Universal Robots PolyScope program: Main.urp

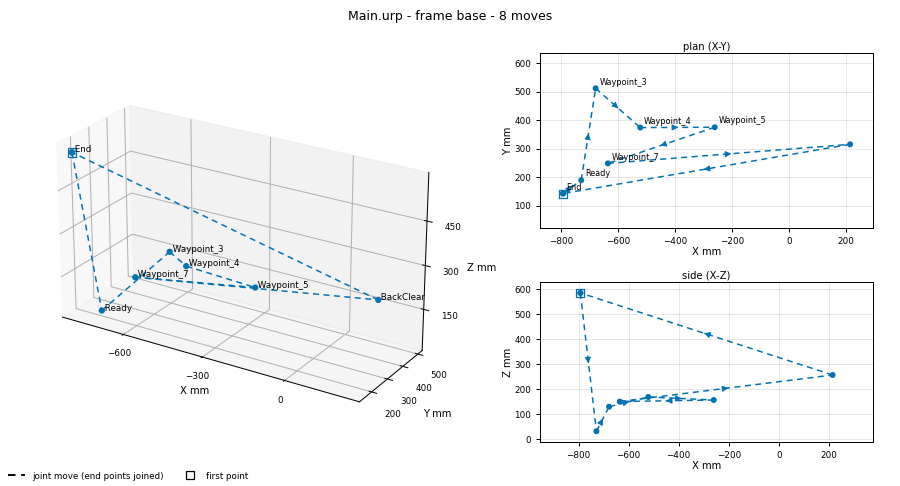
[picture p0: tool path of Main.urp in frame base, 8 of 8 moves have a stored position in this frame; points joined in program order, loops and branches not executed]
Program Main (installation=default directory=/programs/new folder createdIn=5.11.5.1010327 lastSavedIn=5.11.5.1010327 robotSerialNumber=20215500677)
Calibrated DH parameters: a=[0.000204, -0.239222, -0.391845, -0.000001, 0.000022, 0]; d=[0.162722, -355.808559, 353.37206, 2.570385, 0.099741, 0.099629]; alpha=[1.571124, 0.000988, 0.008295, 1.568963, -1.570303, 0]; deltaTheta=[0, -0.973091, 7.204745, 0.05153, 0, 0]
InitVariablesNode variables(variable(name=count, expression=0))
Robot Program (runOnlyOnce=false)
  count := count+1
  Loop Forever
    Wait DigitalInput pin=digital_in[0]; digitalValue=1
    Set DigitalOutput tcp=Dynabrade1; pin=digital_out[1]; digitalValue=1
    MoveJ speed 60 deg/s, acceleration 80 deg/s^2 (useActiveTCP=true) feature=Point_1
      Waypoint End: TCP in base x=-792.986 y=142.126 z=584.824 mm, rx=0.6139 ry=-1.4821 rz=-0.614 rad; joints [333.592, -61.672, 69.104, -187.689, -63.582, 225.626] deg; TCP offset x=0 y=0 z=105 mm, rx=0 ry=0 rz=0 rad; feature pose in base x=-675 y=184.662 z=50 mm, rx=0.0001 ry=0 rz=3.1416 rad
    MoveJ speed 60 deg/s, acceleration 80 deg/s^2 (useActiveTCP=false) tcp=Dynabrade1; feature=Point_1
      Waypoint Ready: TCP in base x=-728.914 y=189 z=32.379 mm, rx=0 ry=-3.1416 rz=0 rad; joints [335.226, -42.704, 75.581, -122.851, -89.577, 245.512] deg; TCP offset x=0 y=0 z=105 mm, rx=0 ry=0 rz=0 rad; feature pose in base x=-728.914 y=189 z=30.379 mm, rx=0 ry=0 rz=3.1416 rad
    Call sandTop
    Call positionFace1
    Call sandFace
    MoveJ speed 60 deg/s, acceleration 80 deg/s^2 (useActiveTCP=true) feature=Point_1
      Waypoint Waypoint_3: TCP in base x=-678.243 y=511.665 z=130.309 mm, rx=-1.5708 ry=0 rz=0 rad; joints [325.381, -29.88, 51.308, -20.942, 145.47, 180.61] deg; TCP offset x=0 y=0 z=105 mm, rx=0 ry=0 rz=0 rad
    Call sandFace
    MoveJ speed 60 deg/s, acceleration 80 deg/s^2 (useActiveTCP=true) feature=Point_1
      Waypoint Waypoint_4: TCP in base x=-521.6 y=373.868 z=169.065 mm, rx=-0.0271 ry=3.1414 rz=-0.0001 rad; joints [312.325, -65.395, 91.797, -116.371, -89.573, 221.581] deg; TCP offset x=0 y=0 z=105 mm, rx=0 ry=0 rz=0 rad
      Waypoint Waypoint_5: TCP in base x=-259.991 y=375 z=156.997 mm, rx=-0.4232 ry=1.5359 rz=-0.398 rad; joints [308.406, -51.401, 88.304, -38.01, -142.187, 238.952] deg; TCP offset x=0 y=0 z=105 mm, rx=0 ry=0 rz=0 rad; feature pose in base x=-585 y=315 z=57 mm, rx=0.0001 ry=0 rz=3.1416 rad
    Call sandFace_1
    URCap Finishing Tool Control (Robotiq_Copilot, Robotiq Inc.) dataModel(FinishingToolStateKey=false, ToolOutputNameKey=digital_out[0], HackTriggeringContributionIsDefinedMethodKey=true)
    MoveJ speed 60 deg/s, acceleration 80 deg/s^2 (useActiveTCP=true) feature=Base
      Waypoint Waypoint_7: TCP in base x=-635.269 y=248.035 z=150.92 mm, rx=-0.4354 ry=3.0052 rz=-0.0196 rad; joints [328.369, -57.223, 80.615, -108.259, -92.837, 222.208] deg; TCP offset x=0 y=0 z=105 mm, rx=0 ry=0 rz=0 rad
    MoveJ speed 60 deg/s, acceleration 80 deg/s^2 (useActiveTCP=true) feature=Point_1
      Waypoint BackClear: TCP in base x=215.017 y=314.968 z=256.959 mm, rx=2.2214 ry=2.2214 rz=0.0002 rad; joints [215.107, -106.327, 122.312, -105.964, -89.576, 215.301] deg; TCP offset x=0 y=0 z=105 mm, rx=0 ry=0 rz=0 rad; feature pose in base x=-585 y=315 z=57 mm, rx=0.0001 ry=0 rz=3.1416 rad
    Call sandBack
    MoveJ speed 60 deg/s, acceleration 80 deg/s^2 (useActiveTCP=true) feature=Point_1
      Waypoint End: TCP in base x=-792.986 y=142.126 z=584.824 mm, rx=0.6139 ry=-1.4821 rz=-0.614 rad; joints [333.592, -61.672, 69.104, -187.689, -63.582, 225.626] deg; TCP offset x=0 y=0 z=105 mm, rx=0 ry=0 rz=0 rad; feature pose in base x=-675 y=184.662 z=50 mm, rx=0.0001 ry=0 rz=3.1416 rad
    Set DigitalOutput tcp=Dynabrade1; pin=digital_out[1]; digitalValue=0
  If count≟20
    Popup Message (haltProgram=false message=change sand paper inputType=Text)
    count := count+1
Event  expression=digital_in[1]≠ True
  Set DigitalOutput tcp=Dynabrade1; pin=digital_out[0]; digitalValue=0
  Set DigitalOutput tcp=Dynabrade1; pin=digital_out[1]; digitalValue=0
  Halt
SubProgram  [hidden by the author, left out]
SubProgram -> sandFace
SubProgram -> sandFace_1
SubProgram -> sandTop
SubProgram -> sandBack
SubProgram sandTop (keepSynchronizedWithDisk=true) programFile=/programs/new folder/sandTop.urp
  MoveL speed 100 mm/s, acceleration 1200 mm/s^2 (useActiveTCP=true) feature=Base
    MoveDirectionNode (selectedDirection=ZPlus) feature=Joint_6_name
      Until TOOL_CONTACT_DETECTION (allowActions=false retraction=0 decelerationAcceleration=3 decelerationAngularAcceleration=34.906585)
  URCap Finishing Tool Control (Robotiq_Copilot, Robotiq Inc.) dataModel(ToolOutputNameKey=digital_out[0], HackTriggeringContributionIsDefinedMethodKey=true)
  Wait Sleep waitTime=2
  URCap Find Surface (Robotiq_Copilot, Robotiq Inc.) dataModel(NodeInitializedKey=true, ZeroSensorBeforeKey=true, WaitForSteadyWrenchOptionKey=false, ls_force=10.0, ls_distance=100.0, ls_speed=5.0, ls_if_distance=false, ls_if_force=false); state(isChildrenLocked=true)
    'Add Stop conditions from the Find Surface node'
  Force Simple feature=Joint_6_name; selection=[0, 0, 1, 0, 0, 0]; wrench=[0, 0, 2, 0, 0, 0]; limitsForce=[0.15, 0.15, 0.15, 1.047198, 1.047198, 1.047198]; limitsMotion=[0.1, 0.1, 0.1, 0.349066, 0.349066, 0.349066]
    MoveL speed 60 mm/s, acceleration 1200 mm/s^2 (useActiveTCP=true) feature=Base
      MoveDirectionNode (selectedDirection=YPlus)
        Until DISTANCE (allowActions=false deceleration=3 distanceNodeType=BLEND) Distance=0.35; motionParameters(blendRadius=0.005)
      MoveDirectionNode (selectedDirection=XPlus)
        Until DISTANCE (allowActions=false deceleration=3 distanceNodeType=BLEND) Distance=0.36; motionParameters(blendRadius=0.005)
      MoveDirectionNode (selectedDirection=YMinus)
        Until DISTANCE (allowActions=false deceleration=3 distanceNodeType=BLEND) Distance=0.35; motionParameters(blendRadius=0.005)
      MoveDirectionNode (selectedDirection=XMinus)
        Until DISTANCE (allowActions=false deceleration=3 distanceNodeType=STOP) Distance=0.36; motionParameters(blendRadius=0.005)
  MoveL speed 60 mm/s, acceleration 1200 mm/s^2 (useActiveTCP=true) feature=Base
    MoveDirectionNode (selectedDirection=ZPlus)
      Until DISTANCE (allowActions=false deceleration=3 distanceNodeType=STOP) Distance=0.025; motionParameters(blendRadius=0)
  URCap Finishing Tool Control (Robotiq_Copilot, Robotiq Inc.) dataModel(ToolOutputNameKey=digital_out[0], FinishingToolStateKey=false, HackTriggeringContributionIsDefinedMethodKey=true)
SubProgram positionFace1 [hidden by the author, left out]
SubProgram sandFace (keepSynchronizedWithDisk=false)
  MoveL speed 250 mm/s, acceleration 1200 mm/s^2 (useActiveTCP=true) feature=Base
    MoveDirectionNode (selectedDirection=ZMinus)
      Until DISTANCE (allowActions=false deceleration=3 distanceNodeType=STOP) Distance=0.072; motionParameters(blendRadius=0)
  MoveL speed 15 mm/s, acceleration 1200 mm/s^2 (useActiveTCP=true) feature=Base
    MoveDirectionNode (selectedDirection=ZPlus) feature=Joint_6_name
      Until TOOL_CONTACT_DETECTION (allowActions=false retraction=0 decelerationAcceleration=3 decelerationAngularAcceleration=34.906585)
    URCap Finishing Tool Control (Robotiq_Copilot, Robotiq Inc.) dataModel(ToolOutputNameKey=digital_out[0], HackTriggeringContributionIsDefinedMethodKey=true)
    Wait Sleep waitTime=2
    URCap Force Control (Robotiq_Copilot, Robotiq Inc.) dataModel(NodeInitializedKey=true, force_x=0, force_y=0, force_mx=0, force_my=0, force_mz=0, limit_x_neg=-100, limit_y_neg=-100, limit_z_neg=-100, limit_x_pos=100, limit_y_pos=100, limit_z_pos=100, limit_mx_neg=-20, limit_my_neg=-20, limit_mz_neg=-20, limit_mx_pos=20, limit_my_pos=20, limit_mz_pos=20, ft_control_x=false, ft_control_y=false, ft_control_mx=false, ft_control_my=false, ft_control_mz=false, stiffness_x=100, stiffness_y=100, stiffness_z_position=100, stiffness_mx=100, stiffness_my=100, stiffness_mz=100, adaptive_stiffness=true, is_force_control_about_actual_position=true, ft_control_z=true, force_z=1, HackTriggeringContributionIsDefinedMethodKey=true, TranslatableFeatureKey=1)
      URCap Force Event (Robotiq_Copilot, Robotiq Inc.) dataModel(NodeInitializedKey=true, NodeTitleKey=Force Event, InteractIfTimeoutOptionKey=false, InteractIfTimeoutNodeInsertedKey=false, InteractTimeoutKey=30, ForceReachedIfTimeoutOptionKey=false, ForceReachedIfTimeoutNodeInsertedKey=false, ForceReachedTimeoutKey=30, IfNotClickedOptionKey=false, IfNotClickedNodeInsertedKey=false, ForceDropRadioButtonKey=true, TorqueDropRadioButtonKey=false, ForceDropKey=10.0, TorqueDropKey=1.0, IsAddSingleTapButtonEnabledKey=true, IsAddDoubleTapButtonEnabledKey=true, AreDuplicatedTapNodesInTreeKey=false, SelectedForceEventKey=2, HackTriggeringContributionIsDefinedMethodKey=true); state(isChildrenLocked=true)
        'Wait until force and torque are reached.'
    MoveDirectionNode (selectedDirection=XPlus) feature=Joint_6_name
      Until DISTANCE (allowActions=false deceleration=3 distanceNodeType=STOP) Distance=0.26; motionParameters(blendRadius=0)
    SuppressedNode
      URCap Find Surface (Robotiq_Copilot, Robotiq Inc.) dataModel(NodeInitializedKey=true, ZeroSensorBeforeKey=true, WaitForSteadyWrenchOptionKey=false, ls_force=10.0, ls_distance=100.0, ls_speed=5.0, ls_if_distance=false, ls_if_force=false); state(isChildrenLocked=true)
        'Add Stop conditions from the Find Surface node'
    SuppressedNode
      Force Simple feature=Joint_6_name; selection=[0, 0, 1, 0, 0, 0]; wrench=[0, 0, 1, 0, 0, 0]; limitsForce=[0.15, 0.15, 0.15, 1.047198, 1.047198, 1.047198]; limitsMotion=[0.1, 0.1, 0.1, 0.349066, 0.349066, 0.349066]
        Placeholder
    URCap Finishing Tool Control (Robotiq_Copilot, Robotiq Inc.) dataModel(FinishingToolStateKey=false, ToolOutputNameKey=digital_out[0], HackTriggeringContributionIsDefinedMethodKey=true)
    MoveDirectionNode (selectedDirection=ZPlus)
      Until DISTANCE (allowActions=false deceleration=3 distanceNodeType=STOP) Distance=0.05; motionParameters(blendRadius=0)
SubProgram sandFace_1 (keepSynchronizedWithDisk=false)
  MoveL speed 250 mm/s, acceleration 1200 mm/s^2 (useActiveTCP=true) feature=Base
    MoveDirectionNode (selectedDirection=ZMinus)
      Until DISTANCE (allowActions=false deceleration=3 distanceNodeType=STOP) Distance=0.072; motionParameters(blendRadius=0)
  MoveL speed 30 mm/s, acceleration 1200 mm/s^2 (useActiveTCP=true) feature=Base
    MoveDirectionNode (selectedDirection=ZPlus) feature=Joint_6_name
      Until TOOL_CONTACT_DETECTION (allowActions=false retraction=0.001 decelerationAcceleration=3 decelerationAngularAcceleration=34.906585)
    URCap Finishing Tool Control (Robotiq_Copilot, Robotiq Inc.) dataModel(ToolOutputNameKey=digital_out[0], HackTriggeringContributionIsDefinedMethodKey=true)
    Wait Sleep waitTime=2
    URCap Force Control (Robotiq_Copilot, Robotiq Inc.) dataModel(NodeInitializedKey=true, force_x=0, force_y=0, force_mx=0, force_my=0, force_mz=0, limit_x_neg=-100, limit_y_neg=-100, limit_z_neg=-100, limit_x_pos=100, limit_y_pos=100, limit_z_pos=100, limit_mx_neg=-20, limit_my_neg=-20, limit_mz_neg=-20, limit_mx_pos=20, limit_my_pos=20, limit_mz_pos=20, ft_control_x=false, ft_control_y=false, ft_control_mx=false, ft_control_my=false, ft_control_mz=false, stiffness_x=100, stiffness_y=100, stiffness_z_position=100, stiffness_mx=100, stiffness_my=100, stiffness_mz=100, adaptive_stiffness=true, is_force_control_about_actual_position=true, ft_control_z=true, force_z=1, HackTriggeringContributionIsDefinedMethodKey=true, TranslatableFeatureKey=1)
      URCap Force Event (Robotiq_Copilot, Robotiq Inc.) dataModel(NodeInitializedKey=true, NodeTitleKey=Force Event, InteractIfTimeoutOptionKey=false, InteractIfTimeoutNodeInsertedKey=false, InteractTimeoutKey=30, ForceReachedIfTimeoutOptionKey=false, ForceReachedIfTimeoutNodeInsertedKey=false, ForceReachedTimeoutKey=30, IfNotClickedOptionKey=false, IfNotClickedNodeInsertedKey=false, ForceDropRadioButtonKey=true, TorqueDropRadioButtonKey=false, ForceDropKey=10.0, TorqueDropKey=1.0, IsAddSingleTapButtonEnabledKey=true, IsAddDoubleTapButtonEnabledKey=true, AreDuplicatedTapNodesInTreeKey=false, SelectedForceEventKey=2, HackTriggeringContributionIsDefinedMethodKey=true); state(isChildrenLocked=true)
        'Wait until force and torque are reached.'
    MoveDirectionNode (selectedDirection=YPlus) feature=Base
      Until DISTANCE (allowActions=false deceleration=3 distanceNodeType=STOP) Distance=0.25; motionParameters(blendRadius=0)
    SuppressedNode
      URCap Find Surface (Robotiq_Copilot, Robotiq Inc.) dataModel(NodeInitializedKey=true, ZeroSensorBeforeKey=true, WaitForSteadyWrenchOptionKey=false, ls_force=10.0, ls_distance=100.0, ls_speed=5.0, ls_if_distance=false, ls_if_force=false); state(isChildrenLocked=true)
        'Add Stop conditions from the Find Surface node'
    SuppressedNode
      Force Simple feature=Joint_6_name; selection=[0, 0, 1, 0, 0, 0]; wrench=[0, 0, 2.5, 0, 0, 0]; limitsForce=[0.15, 0.15, 0.15, 1.047198, 1.047198, 1.047198]; limitsMotion=[0.1, 0.1, 0.1, 0.349066, 0.349066, 0.349066]
        Placeholder
    URCap Finishing Tool Control (Robotiq_Copilot, Robotiq Inc.) dataModel(FinishingToolStateKey=false, ToolOutputNameKey=digital_out[0], HackTriggeringContributionIsDefinedMethodKey=true)
    MoveDirectionNode (selectedDirection=ZPlus)
      Until DISTANCE (allowActions=false deceleration=3 distanceNodeType=STOP) Distance=0.05; motionParameters(blendRadius=0)
SubProgram sandBack (keepSynchronizedWithDisk=true) programFile=/programs/new folder/sandTop.urp
  MoveL speed 100 mm/s, acceleration 600 mm/s^2 (useActiveTCP=true) feature=Base
    MoveDirectionNode (selectedDirection=ZPlus) feature=Joint_6_name
      Until TOOL_CONTACT_DETECTION (allowActions=false retraction=0 decelerationAcceleration=3 decelerationAngularAcceleration=34.906585)
  URCap Finishing Tool Control (Robotiq_Copilot, Robotiq Inc.) dataModel(ToolOutputNameKey=digital_out[0], HackTriggeringContributionIsDefinedMethodKey=true)
  Wait Sleep waitTime=1
  SuppressedNode
    URCap Find Surface (Robotiq_Copilot, Robotiq Inc.) dataModel(NodeInitializedKey=true, WaitForSteadyWrenchOptionKey=false, ls_force=10.0, ls_distance=100.0, ls_speed=5.0, ZeroSensorBeforeKey=true, ls_if_distance=false, ls_if_force=false); state(isChildrenLocked=true)
      'Add Stop conditions from the Find Surface node'
  SuppressedNode
    Force Simple feature=Joint_6_name; selection=[0, 0, 1, 0, 0, 0]; wrench=[0, 0, 1, 0, 0, 0]; limitsForce=[0.15, 0.15, 0.15, 1.047198, 1.047198, 1.047198]; limitsMotion=[0.1, 0.1, 0.1, 0.349066, 0.349066, 0.349066]
      Placeholder
  URCap Force Control (Robotiq_Copilot, Robotiq Inc.) dataModel(NodeInitializedKey=true, force_x=0, force_y=0, force_mx=0, force_my=0, force_mz=0, limit_x_neg=-100, limit_y_neg=-100, limit_z_neg=-100, limit_x_pos=100, limit_y_pos=100, limit_z_pos=100, limit_mx_neg=-20, limit_my_neg=-20, limit_mz_neg=-20, limit_mx_pos=20, limit_my_pos=20, limit_mz_pos=20, ft_control_x=false, ft_control_y=false, ft_control_mx=false, ft_control_my=false, ft_control_mz=false, stiffness_x=100, stiffness_y=100, stiffness_z_position=100, stiffness_mx=100, stiffness_my=100, stiffness_mz=100, adaptive_stiffness=true, is_force_control_about_actual_position=true, HackTriggeringContributionIsDefinedMethodKey=true, ft_control_z=true, force_z=1, TranslatableFeatureKey=1)
    URCap Force Event (Robotiq_Copilot, Robotiq Inc.) dataModel(NodeInitializedKey=true, NodeTitleKey=Force Event, InteractIfTimeoutOptionKey=false, InteractIfTimeoutNodeInsertedKey=false, InteractTimeoutKey=30, ForceReachedIfTimeoutOptionKey=false, ForceReachedIfTimeoutNodeInsertedKey=false, ForceReachedTimeoutKey=30, IfNotClickedOptionKey=false, IfNotClickedNodeInsertedKey=false, ForceDropRadioButtonKey=true, TorqueDropRadioButtonKey=false, ForceDropKey=10.0, TorqueDropKey=1.0, IsAddSingleTapButtonEnabledKey=true, IsAddDoubleTapButtonEnabledKey=true, AreDuplicatedTapNodesInTreeKey=false, SelectedForceEventKey=2, HackTriggeringContributionIsDefinedMethodKey=true); state(isChildrenLocked=true)
      'Wait until force and torque are reached.'
  MoveL speed 45 mm/s, acceleration 1200 mm/s^2 (useActiveTCP=true) feature=Base
    MoveDirectionNode (selectedDirection=YPlus)
      Until DISTANCE (allowActions=false deceleration=3 distanceNodeType=BLEND) Distance=0.35; motionParameters(blendRadius=0.005)
    MoveDirectionNode (selectedDirection=XPlus)
      Until DISTANCE (allowActions=false deceleration=3 distanceNodeType=BLEND) Distance=0.36; motionParameters(blendRadius=0.005)
    MoveDirectionNode (selectedDirection=YMinus)
      Until DISTANCE (allowActions=false deceleration=3 distanceNodeType=BLEND) Distance=0.35; motionParameters(blendRadius=0.005)
    MoveDirectionNode (selectedDirection=XMinus)
      Until DISTANCE (allowActions=false deceleration=3 distanceNodeType=STOP) Distance=0.36; motionParameters(blendRadius=0.005)
  MoveL speed 60 mm/s, acceleration 1200 mm/s^2 (useActiveTCP=true) feature=Base
    MoveDirectionNode (selectedDirection=ZPlus)
      Until DISTANCE (allowActions=false deceleration=3 distanceNodeType=STOP) Distance=0.025; motionParameters(blendRadius=0)
  URCap Finishing Tool Control (Robotiq_Copilot, Robotiq Inc.) dataModel(ToolOutputNameKey=digital_out[0], FinishingToolStateKey=false, HackTriggeringContributionIsDefinedMethodKey=true)
